VAR_GLOBAL CONSTANT
	MAX_INIT_LIST: INT := 64;
END_VAR

(* stored: Version 1.1.0.1, ProductVersion 3.1.4024.10
   GVL GVL_Param: Id {06b257ac-07ca-4920-84f4-18d4d6baa90a} *)
